DATA_BLOCK "dbArchiveEquipExhaust"
{ S7_Optimized_Access := 'TRUE' }
VERSION : 0.8
NON_RETAIN
"fbArchiveEquipExhaust"

BEGIN

END_DATA_BLOCK

